// Mitsubishi GX Works2 project: plc_pj   PLC: Q02/Q02H

// global labels: Global1
VAR_GLOBAL
  공_후 AT X0 : BOOL;
  공_전 AT X1 : BOOL;
  드_상 AT X2 : BOOL;
  드_하 AT X3 : BOOL;
  송_후 AT X4 : BOOL;
  송_전 AT X5 : BOOL;
  배_후 AT X6 : BOOL;
  배_전 AT X7 : BOOL;
  매거진 AT X8 : BOOL;
  비금속 AT X9 : BOOL;
  금속 AT X0A : BOOL;
END_VAR

PROGRAM MAIN
VAR
  테스트 : BOOL;
  송출_전 : BOOL;
  공급_전 : BOOL;
  타이머 : TIMER;
  공급_후 : BOOL;
  가공_전 : BOOL;
  배출_전 : BOOL;
  가공_후 : BOOL;
  배출_후 : BOOL;
  송출_후 : BOOL;
  테스트_종료 : BOOL;
  적색 : BOOL;
  황색 : BOOL;
  녹색 : BOOL;
  황색_테 : BOOL;
  단일회로 : BOOL;
  공급_전1 : BOOL;
  녹색_테 : BOOL;
  공급_후1 : BOOL;
  단일_타이머 : TIMER;
  가공단일작동 : BOOL;
  가공_하1 : BOOL;
  단일_타이머2 : TIMER;
  가공단일해제 : BOOL;
  가공_상1 : BOOL;
  송출_전1 : BOOL;
  송출_후1 : BOOL;
  컨베이어1 : BOOL;
  금속탐지 : BOOL;
  금속판별 : BOOL;
  비금속판별 : BOOL;
  컨베_타이머 : TIMER;
  금속타이머 : TIMER;
  배출_전1 : BOOL;
  배출_후1 : BOOL;
  컨베이어 : BOOL;
  컨베이어스탑 : BOOL;
  단일종료 : BOOL;
END_VAR
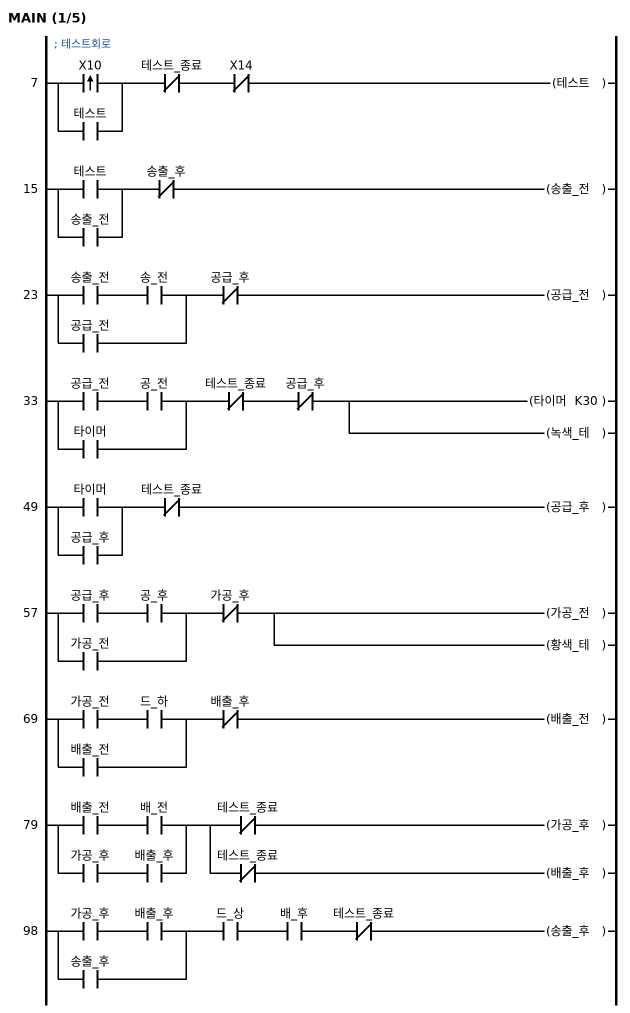
; 테스트회로
7     LDP     X10
      OR      테스트
      ANI     테스트_종료
      ANI     X14
      OUT     테스트
15    LD      테스트
      OR      송출_전
      ANI     송출_후
      OUT     송출_전
23    LD      송출_전
      AND     송_전
      OR      공급_전
      ANI     공급_후
      OUT     공급_전
33    LD      공급_전
      AND     공_전
      OR      타이머
      ANI     테스트_종료
      ANI     공급_후
      OUT     타이머 K30
      OUT     녹색_테
49    LD      타이머
      OR      공급_후
      ANI     테스트_종료
      OUT     공급_후
57    LD      공급_후
      AND     공_후
      OR      가공_전
      ANI     가공_후
      OUT     가공_전
      OUT     황색_테
69    LD      가공_전
      AND     드_하
      OR      배출_전
      ANI     배출_후
      OUT     배출_전
79    LD      배출_전
      AND     배_전
      LD      가공_후
      AND     배출_후
      ORB
      MPS
      ANI     테스트_종료
      OUT     가공_후
      MPP
      ANI     테스트_종료
      OUT     배출_후
98    LD      가공_후
      AND     배출_후
      OR      송출_후
      AND     드_상
      AND     배_후
      ANI     테스트_종료
      OUT     송출_후
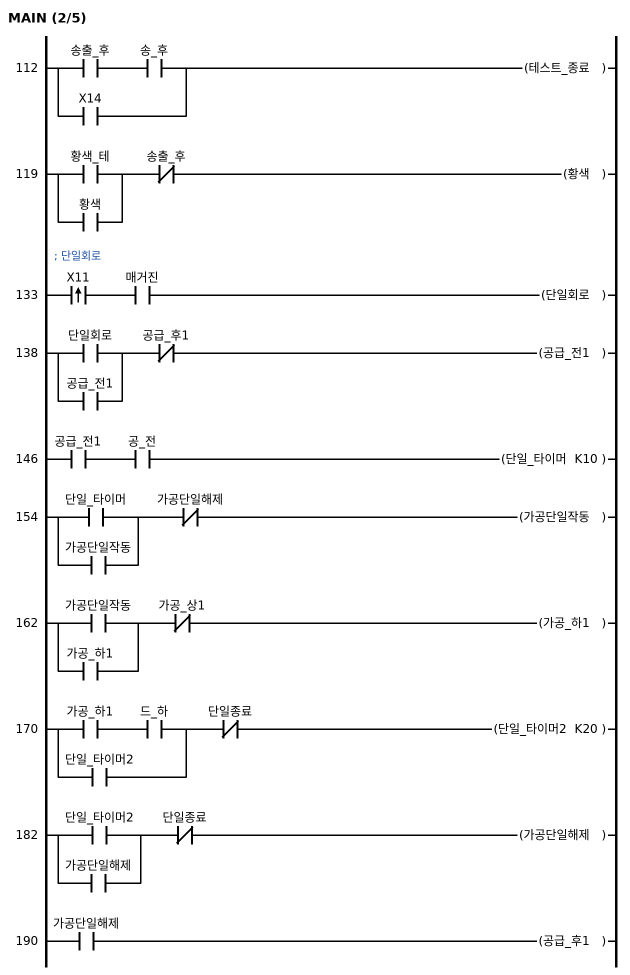
112   LD      송출_후
      AND     송_후
      OR      X14
      OUT     테스트_종료
119   LD      황색_테
      OR      황색
      ANI     송출_후
      OUT     황색
; 단일회로
133   LDP     X11
      AND     매거진
      OUT     단일회로
138   LD      단일회로
      OR      공급_전1
      ANI     공급_후1
      OUT     공급_전1
146   LD      공급_전1
      AND     공_전
      OUT     단일_타이머 K10
154   LD      단일_타이머
      OR      가공단일작동
      ANI     가공단일해제
      OUT     가공단일작동
162   LD      가공단일작동
      OR      가공_하1
      ANI     가공_상1
      OUT     가공_하1
170   LD      가공_하1
      AND     드_하
      OR      단일_타이머2
      ANI     단일종료
      OUT     단일_타이머2 K20
182   LD      단일_타이머2
      OR      가공단일해제
      ANI     단일종료
      OUT     가공단일해제
190   LD      가공단일해제
      OUT     공급_후1
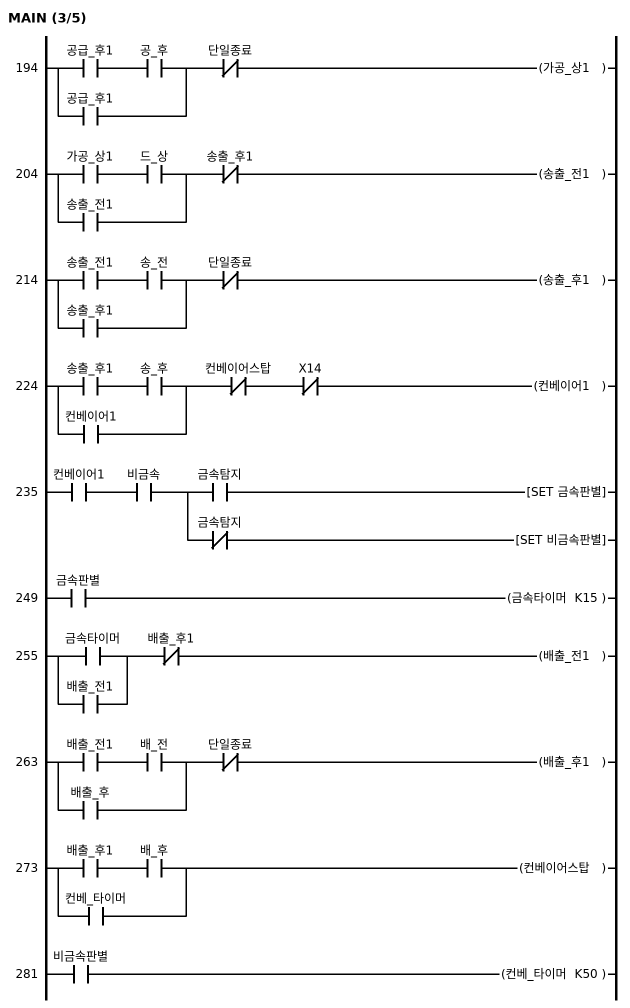
194   LD      공급_후1
      AND     공_후
      OR      공급_후1
      ANI     단일종료
      OUT     가공_상1
204   LD      가공_상1
      AND     드_상
      OR      송출_전1
      ANI     송출_후1
      OUT     송출_전1
214   LD      송출_전1
      AND     송_전
      OR      송출_후1
      ANI     단일종료
      OUT     송출_후1
224   LD      송출_후1
      AND     송_후
      OR      컨베이어1
      ANI     컨베이어스탑
      ANI     X14
      OUT     컨베이어1
235   LD      컨베이어1
      AND     비금속
      MPS
      AND     금속탐지
      SET     금속판별
      MPP
      ANI     금속탐지
      SET     비금속판별
249   LD      금속판별
      OUT     금속타이머 K15
255   LD      금속타이머
      OR      배출_전1
      ANI     배출_후1
      OUT     배출_전1
263   LD      배출_전1
      AND     배_전
      OR      배출_후
      ANI     단일종료
      OUT     배출_후1
273   LD      배출_후1
      AND     배_후
      OR      컨베_타이머
      OUT     컨베이어스탑
281   LD      비금속판별
      OUT     컨베_타이머 K50
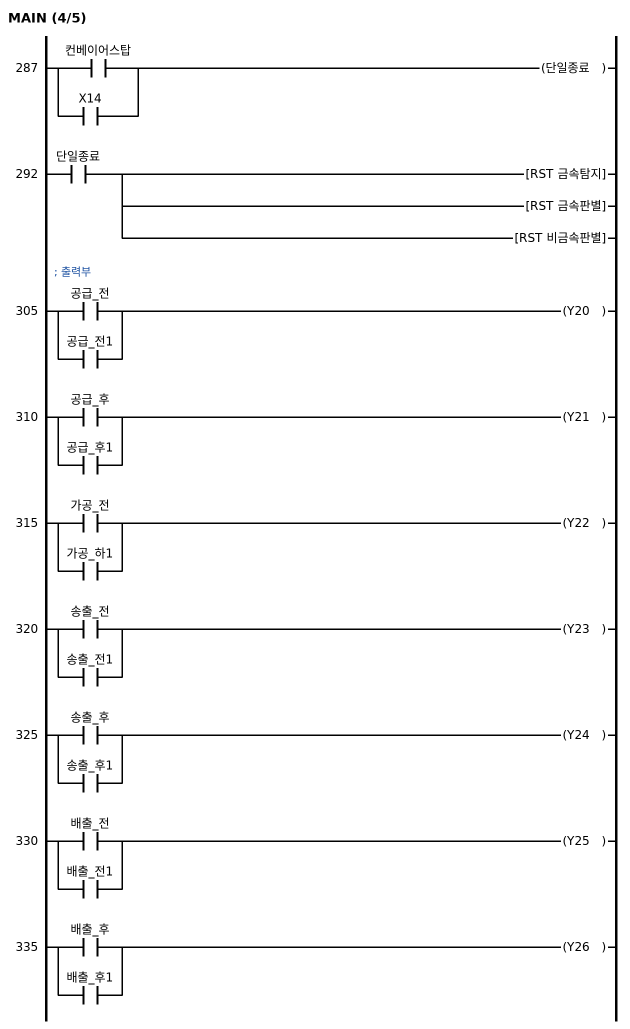
287   LD      컨베이어스탑
      OR      X14
      OUT     단일종료
292   LD      단일종료
      RST     금속탐지
      RST     금속판별
      RST     비금속판별
; 출력부
305   LD      공급_전
      OR      공급_전1
      OUT     Y20
310   LD      공급_후
      OR      공급_후1
      OUT     Y21
315   LD      가공_전
      OR      가공_하1
      OUT     Y22
320   LD      송출_전
      OR      송출_전1
      OUT     Y23
325   LD      송출_후
      OR      송출_후1
      OUT     Y24
330   LD      배출_전
      OR      배출_전1
      OUT     Y25
335   LD      배출_후
      OR      배출_후1
      OUT     Y26
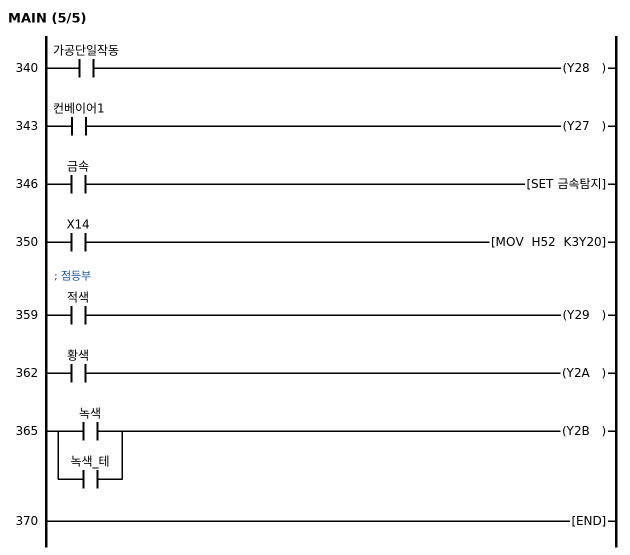
340   LD      가공단일작동
      OUT     Y28
343   LD      컨베이어1
      OUT     Y27
346   LD      금속
      SET     금속탐지
350   LD      X14
      MOV     H52 K3Y20
; 점등부
359   LD      적색
      OUT     Y29
362   LD      황색
      OUT     Y2A
365   LD      녹색
      OR      녹색_테
      OUT     Y2B
370   END
END_PROGRAM
